PROGRAM MAIN
VAR
	stTank1 : ST_Tank := (nId := 101,fTemperature := 80.3, fLevel := 80, bAlarm := FALSE );
	stTank2 : ST_Tank  := (nId := 102,fTemperature := 72.5, fLevel := 70, bAlarm := FALSE );
	stTank3 : ST_Tank  := (nId := 103,fTemperature := 90.8, fLevel := 90, bAlarm := FALSE );
	
	fbController : FB_TankController;
	iTankController : I_TankController;
	
	bStart : BOOl;
END_VAR

IF bStart THEN
	fbController(stTank := stTank1);
	bStart := FALSE;
END_IF

END_PROGRAM

(* stored: Version 1.1.0.1, ProductVersion 3.1.4024.16
   POU MAIN: Id {6b8a6ca2-acf4-4660-828c-fe5694732b70}, SpecialFunc None *)
